FUNCTION_BLOCK CONCAT_QUERY
  {SET_ATTRIBUTE(OpcUa, SERVICE)}
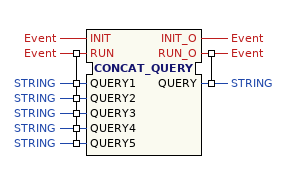
  EVENT_INPUT
    INIT;
    RUN WITH QUERY1, QUERY2, QUERY3, QUERY4, QUERY5; {SET_ATTRIBUTE(OpcUa, Method)}
  END_EVENT
  EVENT_OUTPUT
    INIT_O;
    RUN_O WITH QUERY;
  END_EVENT
  VAR_INPUT
    QUERY1 : STRING;
    QUERY2 : STRING;
    QUERY3 : STRING;
    QUERY4 : STRING;
    QUERY5 : STRING;
  END_VAR
  VAR_OUTPUT
    QUERY : STRING;
  END_VAR
END_FUNCTION_BLOCK
